PROGRAM MAIN
VAR
	rPosSenDis_mm : REAL;
	rPosSenDis_inch : REAL;
END_VAR

GVL.rCurrent_Input1_EU := GVL.nCurrent_Input1 * 16.0/(26300.0); //16 mA/(range of DAQ resolution)
rPosSenDis_mm := (GVL.rCurrent_Input1_EU - 3.92) / 0.01260;//mm displacement
rPosSenDis_inch := f_mmToInch(rPosSenDis_mm);

END_PROGRAM

(* stored: Version 1.1.0.1, ProductVersion 3.1.4024.12
   POU MAIN: Id {5bb984b1-30f5-48aa-9dca-5dbeed0d3db1}, SpecialFunc None *)
